Staubli VAL3: getSize.pgx

public program getSize(num& x_nSize[] (dimensions=1))
  local num i
  local num l_nSize
  local bool l_bFound
  local string l_sEmpty
  local string l_sPath
  local string l_sType
  local string l_sKey
  local string l_sItem
begin
  // give back the size to trajectory field
  x_nSize=size(saveProg:pProg)
end
